INTERFACE I_Sequence

END_INTERFACE

(* stored: Version 1.1.0.1, ProductVersion 3.1.4024.12
   Itf I_Sequence: Id {59568bd8-d8a4-402f-82c8-f495286ce9cc} *)
